// TwinCAT 3 PLC project EFillerv1
// ProgramVersion: 3.1.4023.0
// libraries:
//   Tc2_Standard, * (Beckhoff Automation GmbH)
//   Tc2_System, * (Beckhoff Automation GmbH)
//   Tc3_Module, * (Beckhoff Automation GmbH)
// project tree:
//   DUTs/ ActInputs.TcDUT, ActOutputs.TcDUT, Buttons.TcDUT, Flags.TcDUT
//   / PlcTask.TcTTO
//   POUs/0. Ignition/ ButtonCheck.TcPOU
//   POUs/1. Actuators/ Gripper.TcPOU, HorizontalAct.TcPOU, VerticalAct.TcPOU
//   POUs/3. Flags/ CycleCount.TcPOU
//   POUs/4. FSM/ Wrapper.TcPOU
//   POUs/ MAIN.TcPOU
//   POUs/2. Sensors/ CellSensor.TcPOU

CONFIGURATION EFillerv1
    RESOURCE PLC ON TwinCAT3
        TASK PlcTask(INTERVAL := T#10ms, PRIORITY := 22);
        PROGRAM MAIN WITH PlcTask : MAIN;
    END_RESOURCE
END_CONFIGURATION

// ---- DUTs/ActInputs.TcDUT
TYPE ActInputs :
STRUCT
	Extended 	: BOOL;
	Retracted 	: BOOL;
	Raised 		: BOOL;
	Lowered 	: BOOL;
	Opened 		: BOOL;
	Closed 		: BOOL;

END_STRUCT
END_TYPE

// ---- DUTs/ActOutputs.TcDUT
TYPE ActOutputs :
STRUCT
	Extend 	: BOOL;
	Raise 	: BOOL;
	Close 	: BOOL;

END_STRUCT
END_TYPE

// ---- DUTs/Buttons.TcDUT
TYPE Buttons :
STRUCT
	Start : BOOL;
	EStop : BOOL;
	Reset : BOOL;
END_STRUCT
END_TYPE

// ---- DUTs/Flags.TcDUT
TYPE Flags :
STRUCT
	PlaceReady	: BOOL;
	PartReady	: BOOL;
	Picked		: Bool;
END_STRUCT
END_TYPE

// ---- POUs/MAIN.TcPOU
PROGRAM MAIN
VAR
	Station : Wrapper;
	
	ActInputs	: ActInputs;
	ActOutputs	: ActOutputs;
	Buttons		: Buttons;
	Flags		: Flags;
END_VAR

Station(ActInputs 	:= ActInputs,
		ActOutputs	=> ActOutputs,
		Buttons		:= Buttons,
		Flags		=> Flags);

END_PROGRAM

// ---- POUs/4. FSM/Wrapper.TcPOU
FUNCTION_BLOCK Wrapper
VAR_INPUT
	ActInputs   : ActInputs;
	Buttons		: Buttons;  
END_VAR
VAR_OUTPUT
	ActOutputs	: ActOutputs;
	Flags		: Flags;
END_VAR
VAR	
	ButtonCheck		: ButtonCheck;

	Gripper			: Gripper;
	HorizontalAct	: HorizontalAct;
	VerticalAct		: VerticalAct;
	CellSensor		: CellSensor;
	CycleCount		: CycleCount;
END_VAR

METHOD mMap : BOOL
VAR_INPUT
END_VAR
/////// Inputs //////////
Gripper.pClosed		:= ActInputs.Closed;
Gripper.pOpened		:= ActInputs.Opened;
HorizontalAct.pExtended		:= ActInputs.Extended;
HorizontalAct.pRetracted	:= ActInputs.Retracted;
VerticalAct.pLowered	:= ActInputs.Lowered;
VerticalAct.pRaised		:= ActInputs.Raised;
ButtonCheck.pEStop	:= Buttons.EStop;
ButtonCheck.pReset	:= Buttons.Reset;
ButtonCheck.pStart	:= Buttons.Start;

/////// Outputs //////////
ActOutputs.Close 	:= Gripper.pClose;
ActOutputs.Extend	:= HorizontalAct.pExtend;
ActOutputs.Raise	:= VerticalAct.pRaise;
Flags.PartReady 	:= CellSensor.pFeeded;
Flags.PlaceReady	:= CellSensor.pOKtoRelase;
Flags.Picked		:= CycleCount.pPicked;
END_METHOD

END_FUNCTION_BLOCK

// ---- POUs/0. Ignition/ButtonCheck.TcPOU
FUNCTION_BLOCK ButtonCheck
VAR
	Start 	: BOOL;
	EStop 	: BOOL;
	Reset	: BOOL;
	
END_VAR

METHOD mEStop : BOOL
VAR_INPUT
END_VAR
//pEStop := Buttons.EStop := TRUE; (Faulty)
pEStop := TRUE;
END_METHOD

METHOD mReset : BOOL
VAR_INPUT
END_VAR
pReset := TRUE;
END_METHOD

METHOD mStart : BOOL
VAR_INPUT
END_VAR
pStart := TRUE;
END_METHOD

PROPERTY pEStop : BOOL
GET
pEStop := EStop;
END_GET
SET
EStop := pEStop;
END_SET
END_PROPERTY

PROPERTY pReset : BOOL
GET
pReset := Reset;
END_GET
SET
Reset := pReset;
END_SET
END_PROPERTY

PROPERTY pStart : BOOL
GET
pStart := Start;
END_GET
SET
Start := pStart;
END_SET
END_PROPERTY

END_FUNCTION_BLOCK

// ---- POUs/1. Actuators/Gripper.TcPOU
FUNCTION_BLOCK Gripper
VAR
	Close	: BOOL;
	Closed	: BOOL;
	Opened 	: BOOL;
END_VAR

METHOD mClose : BOOL
VAR_INPUT
END_VAR
//IF ActInputs.Opened AND Flags.PartReady THEN (Faulty)
//	Close := ActOutputs.Close := TRUE;
//END_IF

Close := TRUE;
END_METHOD

METHOD mClosed : BOOL
VAR_INPUT
END_VAR
END_METHOD

METHOD mOpened : BOOL
VAR_INPUT
END_VAR
END_METHOD

PROPERTY pClose : BOOL
GET
pClose := Close;
END_GET
SET
Close := pClose;
END_SET
END_PROPERTY

PROPERTY pClosed : BOOL
GET
pClosed := Closed;
END_GET
SET
Closed := pClosed;
END_SET
END_PROPERTY

PROPERTY pOpened : BOOL
GET
END_GET
SET
END_SET
END_PROPERTY

END_FUNCTION_BLOCK

// ---- POUs/1. Actuators/HorizontalAct.TcPOU
FUNCTION_BLOCK HorizontalAct
VAR_INPUT
END_VAR
VAR_OUTPUT
	Extend		: BOOL;
	Extended	: BOOL;
	Retracted 	: BOOL;
	
END_VAR
VAR
END_VAR

METHOD mExtend : BOOL
VAR_INPUT
END_VAR
//IF ActInputs.Retracted AND Flags.PartReady THEN (Faulty)
//	Extend	:= ActOutputs.Extend := TRUE;
//END_IF
Extend	:= TRUE;
END_METHOD

METHOD mExtended : BOOL
VAR_INPUT
END_VAR
END_METHOD

METHOD mRetracted : BOOL
VAR_INPUT
END_VAR
END_METHOD

PROPERTY pExtend : BOOL
GET
pExtend	:= Extend;
END_GET
SET
Extend	:= pExtend;
END_SET
END_PROPERTY

PROPERTY pExtended : BOOL
GET
pExtended := Extended;
END_GET
SET
Extended := pExtended;
END_SET
END_PROPERTY

PROPERTY pRetracted : BOOL
GET
pRetracted := Retracted;
END_GET
SET
Retracted := pRetracted;
END_SET
END_PROPERTY

END_FUNCTION_BLOCK

// ---- POUs/1. Actuators/VerticalAct.TcPOU
FUNCTION_BLOCK VerticalAct
VAR_INPUT
END_VAR
VAR_OUTPUT
	Raise	: BOOL;
	Raised	: BOOL;
	Lowered	: BOOL;
	
END_VAR
VAR
END_VAR

METHOD mLowered : BOOL
VAR_INPUT
END_VAR
END_METHOD

METHOD mRaise : BOOL
VAR_INPUT
END_VAR
//IF ActInputs.Lowered AND ActInputs.Closed THEN (Faulty)
//	Raise	:= ActOutputs.Raise := TRUE;
//END_IF

Raise	:= TRUE;
END_METHOD

METHOD mRaised : BOOL
VAR_INPUT
END_VAR
END_METHOD

PROPERTY pLowered : BOOL
GET
pLowered := Lowered;
END_GET
SET
Lowered := pLowered;
END_SET
END_PROPERTY

PROPERTY pRaise : BOOL
GET
pRaise	:= Raise;
END_GET
SET
Raise	:= pRaise;
END_SET
END_PROPERTY

PROPERTY pRaised : BOOL
GET
pRaised := Raised;
END_GET
SET
Raised := pRaised;
END_SET
END_PROPERTY

END_FUNCTION_BLOCK

// ---- POUs/2. Sensors/CellSensor.TcPOU
FUNCTION_BLOCK CellSensor
VAR
	OKtoRelase 	: BOOL;
	Feeded	: BOOL;
	
END_VAR

METHOD mFeeded : BOOL
VAR_INPUT
END_VAR
Feeded := True;
END_METHOD

METHOD mOKtoRelase : BOOL
VAR_INPUT
END_VAR
OKtoRelase := TRUE;
END_METHOD

PROPERTY pFeeded : BOOL
GET
pFeeded := Feeded;
END_GET
SET
Feeded := pFeeded;
END_SET
END_PROPERTY

PROPERTY pOKtoRelase : BOOL
GET
pOKtoRelase := OKtoRelase;
END_GET
SET
OKtoRelase := pOKtoRelase;
END_SET
END_PROPERTY

END_FUNCTION_BLOCK

// ---- POUs/3. Flags/CycleCount.TcPOU
FUNCTION_BLOCK CycleCount
VAR
	Picked : BOOL;
	
END_VAR

METHOD mPicked : BOOL
VAR_INPUT
END_VAR
Picked := TRUE;
END_METHOD

PROPERTY pPicked : BOOL
GET
pPicked := Picked;
END_GET
SET
Picked := pPicked;
END_SET
END_PROPERTY

END_FUNCTION_BLOCK
